TYPE stInOuts :
STRUCT
	bOverCurrent		AT %I*	: BOOL;			//Przekroczony prąd
	bSafety				AT %I*	: BOOL;			//Obsługa safety
	bPowerON			AT %Q*	: BOOL;			//Załączenie zasilania
	bFanON				AT %Q*	: BOOL;			//Załączenie wentylatora
	bPressureIn			AT %Q*	: BOOL;			//Dobicie ciśnienia do ustalonwej na manometrze wartości
	bBottle40l			AT %Q*	: BOOL;			//Załączenie testu z butlą 40l
	bEjectPresure		AT %Q*	: BOOL;			//Zrzucenie ciśnienia z butli 1l
	bEjectPresure40		AT %Q*	: BOOL;			//Zrzucenie ciśnmienia z butli 40l
	
	iPressureRaw		AT %I* 	: INT;			//Surowa wartość ciśnienia
	iVoltageRaw			AT %I*	: INT;			//Surowa wartość napięcia
	iCurrentRaw			AT %I*	: INT;			//Surowa wartość prądu
	
	rPressure			 		: REAL;			//Wartość ciśnienia
	rVoltage					: REAL;			//Wartość napięcia
	rCurrent					: REAL;			//Wartość prądu
	rTemperature				: REAL;			//Wartość temperatury
	iTemperature		AT %I*	: INT;			//Wartość temperatury
END_STRUCT
END_TYPE

(* stored: Version 1.1.0.1, ProductVersion 3.1.4024.12
   DUT stInOuts: Id {7fe2b391-15c8-427d-b951-00317dc5b688} *)
